(* Schneider Machine Expert - Basic project Tank_Level_Safe_v12, file version 3.0.0.0 *)
(* ProjectInformations: Name=New project *)

HARDWARE
  Cpu 0: TM221CE24T
  ModuleExtensionObject 0: TM3AI4/G
  EthernetConfiguration: NetworkName=M221, IpAllocationMode=FixedAddress, IpAddress=0.0.0.0, SubnetMask=0.0.0.0
  SerialLineConfiguration: Baud=Baud19200, Parity=ParityEven, DataBits=DataBits8, StopBits=StopBits1, PhysicalMedium=PhysicalMediumRs485, TransmissionMode=TransmissionModeModbusRtu, SlaveId=1, Addressing=SlaveAddressing
  MastTask: UsePeriodScanMode=false, PeriodScan=100
  FastTask: Period=255
  CpuBehavior: StartingMode=StartAsPreviousState, AutoSaveRamOnEeprom=true, WatchdogPeriod=250

SYMBOLS  (address, symbol, comment, settings)
  %IW1.0    TANK_LEVEL  [Type=Type_4_20mA, Scope=Scope_Customized, Minimum=300, Maximum=3000]

POU New POU
  (* SectionNumber=0 *)

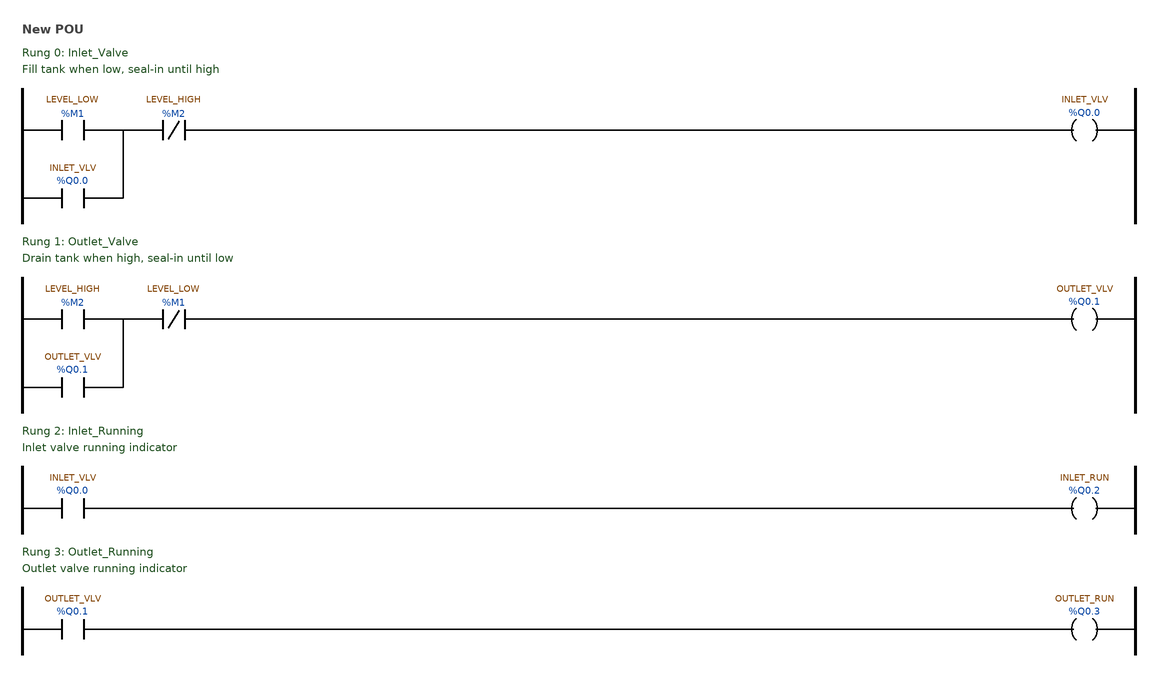

// Rung 0: Inlet_Valve
// Fill tank when low, seal-in until high
  LD %M1
  OR %Q0.0
  ANDN %M2
  ST %Q0.0
  // as ST:
  //   %Q0.0 := (%M1 OR %Q0.0) AND NOT %M2;

// Rung 1: Outlet_Valve
// Drain tank when high, seal-in until low
  LD %M2
  OR %Q0.1
  ANDN %M1
  ST %Q0.1
  // as ST:
  //   %Q0.1 := (%M2 OR %Q0.1) AND NOT %M1;

// Rung 2: Inlet_Running
// Inlet valve running indicator
  LD %Q0.0
  ST %Q0.2
  // as ST:
  //   %Q0.2 := %Q0.0;

// Rung 3: Outlet_Running
// Outlet valve running indicator
  LD %Q0.1
  ST %Q0.3
  // as ST:
  //   %Q0.3 := %Q0.1;
